# EPICS substitutions: plcApp_IntLock/exampleApp/Db/user.substitutions
# Example substitutions file

file "db/dbExample1.db" {
    { user = "jiangbo" }
}

file db/dbExample2.db {
    pattern { user, no, scan }
        { "jiangbo", 1, "1 second" }
        { "jiangbo", 2, "2 second" }
        { "jiangbo", 3, "5 second" }
}
